// TwinCAT 3 PLC project Tc3_IoLink_Samples
// ProgramVersion: 3.1.4023.0
// libraries:
//   Tc2_Standard, * (Beckhoff Automation GmbH)
//   Tc2_System, * (Beckhoff Automation GmbH)
//   Tc3_IoLink, * (Beckhoff Automation GmbH)
//   Tc3_Module, * (Beckhoff Automation GmbH)
// project tree:
//   GVLs/ GVL_IO.TcGVL
//   / PlcTask.TcTTO
//   POUs/Samples/ FB_Sample_01_IolRead.TcPOU, FB_Sample_03_IolSlave.TcPOU, FB_Sample_02_IolWrite.TcPOU, FB_Sample_04_IolStdVarSlave.TcPOU, FB_Sample_06_IdentificationAndDiagnosis.TcPOU, FB_Sample_07_MeasurementDataChannel.TcPOU
//   POUs/ MAIN.TcPOU
// real-time tasks:
//   TASK PlcTask: cycle T#10ms, priority 20, ADS port 350
// I/O:
//   DEVICE Device 1 (EtherCAT), AmsNetId 192.168.178.79.2.1
//     Term 1 (EK1100) [EK1100 EtherCAT Coupler (2A E-Bus)]
//       Term 2 (EL6224) [EL6224 (IO Link Master)]
// variable links:
//   Tc3_IoLink_Samples/Tc3_IoLink_Samples Instance <-> Device 1 (EtherCAT)/Term 1 (EK1100)/Term 2 (EL6224)
//     PlcTask Inputs/GVL_IO.nTerm2Port{1..4}State <-> DeviceState Inputs/State Ch{1..4}  (4 links)
//     PlcTask Inputs/GVL_IO.sTerm2AmsNetId <-> InfoData/AoeNetId

CONFIGURATION Tc3_IoLink_Samples
    RESOURCE PLC ON TwinCAT3
        TASK PlcTask(INTERVAL := T#10ms, PRIORITY := 20);
        PROGRAM MAIN WITH PlcTask : MAIN;
    END_RESOURCE
END_CONFIGURATION

// ---- GVLs/GVL_IO.TcGVL
{attribute 'qualified_only'}
VAR_GLOBAL
	sTerm2AmsNetId 	AT%I*			: AMSNETID;
	
	nTerm2EPI1008					: E_IolPort := E_IolPort.Port1;
	nTerm2EPI2008					: E_IolPort := E_IolPort.Port2;
	nTerm2EPI3174					: E_IolPort := E_IolPort.Port3;

	nTerm2Port1State 	AT%I*		: USINT;
	nTerm2Port2State 	AT%I*		: USINT;
	nTerm2Port3State 	AT%I*		: USINT;
	nTerm2Port4State 	AT%I*		: USINT;
END_VAR

// ---- POUs/MAIN.TcPOU
PROGRAM MAIN
VAR
	fbSample_01_IolRead 					: FB_Sample_01_IolRead;
	fbSample_02_IolWrite 					: FB_Sample_02_IolWrite;
	fbSample_03_IolSlave 					: FB_Sample_03_IolSlave;
	fbSample_04_IolStdVarSlave 				: FB_Sample_04_IolStdVarSlave;
	fbSample_06_IdentificationAndDiagnosis	: FB_Sample_06_IdentificationAndDiagnosis;
	fbSample_07_MeasurementDataChannel		: FB_Sample_07_MeasurementDataChannel;
END_VAR


fbSample_01_IolRead(); 		
fbSample_02_IolWrite();	
fbSample_03_IolSlave(); 
fbSample_04_IolStdVarSlave();
fbSample_06_IdentificationAndDiagnosis();

END_PROGRAM

// ---- POUs/Samples/FB_Sample_01_IolRead.TcPOU
FUNCTION_BLOCK FB_Sample_01_IolRead
VAR_INPUT
	bExecute				: BOOL := FALSE;
END_VAR
VAR_OUTPUT
	bBusy					: BOOL := FALSE;
	bDone					: BOOL := FALSE;
	bError					: BOOL := FALSE;
	nAdsError				: E_AdsErr := E_AdsErr.NOERR;
	nIolError				: E_IolError := E_IolError.NoError;
	sErrorTxt				: STRING(255) := '';
	sApplicationTag			: STRING(32) := '';
END_VAR
VAR
	bExecuteOld				: BOOL;
	nState					: INT := 0;
	fbIolRead 				: FB_IolRead;
END_VAR

////
// Execute/Busy State Machine
//
IF bExecute AND NOT bExecuteOld AND NOT bBusy THEN
	bBusy := TRUE;
	nState := 10;	// READ
ELSIF NOT bExecute THEN
	bBusy := FALSE;
	bError := FALSE;
	bDone := FALSE;
	nAdsError := E_AdsErr.NOERR;
	nIolError := E_IolError.NoError;
	sErrorTxt := '';
END_IF
bExecuteOld := bExecute;

////
// FB State Machine
//
CASE nState OF
// IDLE
0:;
// READ
10:
	sApplicationTag := '';
	
	fbIolRead(bExecute := FALSE);
	fbIolRead.sNetId := F_CreateAmsNetId(GVL_IO.sTerm2AmsNetId);
	fbIolRead.nIolPort := E_IolPort.Port1;
	fbIolRead.pDSTBuf := ADR(sApplicationTag);
	fbIolRead.cbBufLen := 32;
	fbIolRead.nIndex := 16#18; 
	fbIolRead.nSubindex := 0;
	fbIolRead.bExecute := TRUE;
	
	nState := 20; // WAIT_FOR_DONE 
	
// WAIT_FOR_DONE
20:
	IF fbIolRead.bDone THEN
		bDone := TRUE;
		bBusy := FALSE;
		nState := 0; // IDLE
	END_IF 
END_CASE

////
// call FBs
//
fbIolRead();

////
// Error Handling
//
IF NOT bError AND bBusy THEN
	IF fbIolRead.bError THEN
		nState := 0;
		bBusy := FALSE;
		bError := TRUE;
		nAdsError := fbIolRead.nAdsError;
		nIolError := fbIolRead.nIolError;
		sErrorTxt := F_IolGetErrorTxt(fbIolRead.hresult);
	END_IF
END_IF

END_FUNCTION_BLOCK

// ---- POUs/Samples/FB_Sample_02_IolWrite.TcPOU
FUNCTION_BLOCK FB_Sample_02_IolWrite
VAR_INPUT
	bExecute				: BOOL := FALSE;
	sApplicationTag			: STRING(32) := '';
END_VAR
VAR_OUTPUT
	bBusy					: BOOL := FALSE;
	bDone					: BOOL := FALSE;
	bError					: BOOL := FALSE;
	nAdsError				: E_AdsErr := E_AdsErr.NOERR;
	nIolError				: E_IolError := E_IolError.NoError;
	sErrorTxt				: STRING(255) := '';
END_VAR
VAR
	bExecuteOld				: BOOL;
	nState					: INT := 0;
	fbIolWrite 				: FB_IolWrite;
END_VAR

////
// Execute/Busy State Machine
//
IF bExecute AND NOT bExecuteOld AND NOT bBusy THEN
	bBusy := TRUE;
	nState := 10;	// WRITE
ELSIF NOT bExecute THEN
	bBusy := FALSE;
	bError := FALSE;
	bDone := FALSE;
	nAdsError := E_AdsErr.NOERR;
	nIolError := E_IolError.NoError;
	sErrorTxt := '';
END_IF
bExecuteOld := bExecute;


////
// FB State Machine
//
CASE nState OF
	
// IDLE
0:;

// WRITE
10:	
	fbIolWrite(bExecute := FALSE);
	fbIolWrite.sNetId := F_CreateAmsNetId(GVL_IO.sTerm2AmsNetId);
	fbIolWrite.nIolPort := GVL_IO.nTerm2EPI1008;
	fbIolWrite.pSRCBuf := ADR(sApplicationTag);
	fbIolWrite.cbBufLen := 32;
	fbIolWrite.nIndex := 16#18;
	fbIolWrite.nSubindex := 0;
	fbIolWrite.bExecute := TRUE;
	
	nState := 20; // WAIT_FOR_DONE 
	
// WAIT_FOR_DONE
20:
	IF fbIolWrite.bDone THEN
		bDone := TRUE;
		bBusy := FALSE;
		nState := 0; // IDLE
	END_IF 
END_CASE


////
// call FBs
//
fbIolWrite();

////
// Error Handling
//
IF NOT bError AND bBusy THEN
	IF fbIolWrite.bError THEN
		nState := 0;
		bBusy := FALSE;
		bError := TRUE;
		nAdsError := fbIolWrite.nAdsError;
		nIolError := fbIolWrite.nIolError;
		sErrorTxt := F_IolGetErrorTxt(fbIolWrite.hresult);
	END_IF
END_IF

END_FUNCTION_BLOCK

// ---- POUs/Samples/FB_Sample_03_IolSlave.TcPOU
FUNCTION_BLOCK FB_Sample_03_IolSlave
VAR_INPUT
	bExecute				: BOOL := FALSE;
	sApplicationTag			: STRING(32) := '';
END_VAR
VAR_OUTPUT
	bBusy					: BOOL := FALSE;
	bDone					: BOOL := FALSE;
	bError					: BOOL := FALSE;
	nAdsError				: E_AdsErr := E_AdsErr.NOERR;
	nIolError				: E_IolError := E_IolError.NoError;
	sErrorTxt				: STRING(255) := '';
END_VAR
VAR
	bExecuteOld				: BOOL;
	nState					: INT := 0;
	fbIolSlave 				: FB_IolSlave;
	bInitDone				: BOOL := FALSE;
	hr						: HRESULT;
	sApplicationTagRead		: STRING(32) := '';
	sData					: STRING;
END_VAR

////
// Init
//
IF NOT bInitDone THEN
	bInitDone := TRUE;
	fbIolSlave.MasterAoeNetId := F_CreateAmsNetId(GVL_IO.sTerm2AmsNetId);
	fbIolSlave.Port := GVL_IO.nTerm2EPI1008;
	fbIolSlave.Name := 'EPI1008';
END_IF

////
// Execute/Busy State Machine
//
IF bExecute AND NOT bExecuteOld AND NOT bBusy THEN
	bBusy := TRUE;
	nState := 10;	// WRITE
ELSIF NOT bExecute THEN
	bBusy := FALSE;
	bError := FALSE;
	bDone := FALSE;
	nAdsError := E_AdsErr.NOERR;
	nIolError := E_IolError.NoError;
	sErrorTxt := '';
END_IF
bExecuteOld := bExecute;


////
// FB State Machine
//
CASE nState OF
	
// IDLE
0:;

// WRITE
10:
	hr := fbIolSlave.Write(16#0018, 0, ADR(sApplicationTag), 32);
	IF NOT F_IolIsBusy(hr) THEN
		IF FAILED(hr) THEN
			bBusy := FALSE;
			bError := TRUE;
			sErrorTxt := fbIolSlave.ErrorTxt;
			nAdsError := F_IolGetAdsError(hr);
			nIolError := F_IolGetIolError(hr);
			nState := 0; // IDLE;
		ELSE
			nState := 20; // READ;
		END_IF
	END_IF
	
// READ
20:
	hr := fbIolSlave.Read(16#0018, 16#00, ADR(sApplicationTagRead), 32);
	IF NOT F_IolIsBusy(hr) THEN
		IF FAILED(hr) THEN
			bBusy := FALSE;
			bError := TRUE;
			sErrorTxt := fbIolSlave.ErrorTxt;
			nAdsError := F_IolGetAdsError(hr);
			nIolError := F_IolGetIolError(hr);
			nState := 0; // IDLE;
		ELSE
			nState := 30; // CHECK;
		END_IF
	END_IF
	
// CHECK
30:
	IF sApplicationTag <> sApplicationTagRead THEN
		bBusy := FALSE;
		bError := TRUE;
		sErrorTxt := 'sApplicationTag and sApplicationTagRead are not equal!';
	ELSE
		bBusy := FALSE;
		bDone := TRUE;
		nState := 0;
	END_IF
END_CASE


////
// call FBs
//
fbIolSlave();

END_FUNCTION_BLOCK

// ---- POUs/Samples/FB_Sample_04_IolStdVarSlave.TcPOU
FUNCTION_BLOCK FB_Sample_04_IolStdVarSlave
VAR_INPUT
	bExecute				: BOOL := FALSE;
	sApplicationTag			: STRING(32) := '';
END_VAR
VAR_OUTPUT
	bBusy					: BOOL := FALSE;
	bDone					: BOOL := FALSE;
	bError					: BOOL := FALSE;
	nAdsError				: E_AdsErr := E_AdsErr.NOERR;
	nIolError				: E_IolError := E_IolError.NoError;
	sErrorTxt				: STRING(255) := '';
END_VAR
VAR
	bExecuteOld				: BOOL;
	nState					: INT := 0;
	fbIolSlave 				: FB_IolStdVarSlave;
	bInitDone				: BOOL := FALSE;
	hr						: HRESULT;
	sApplicationTagRead		: STRING(32) := '';
END_VAR

////
// Init
//
IF NOT bInitDone THEN
	bInitDone := TRUE;
	fbIolSlave.MasterAoeNetId := F_CreateAmsNetId(GVL_IO.sTerm2AmsNetId);
	fbIolSlave.Port := GVL_IO.nTerm2EPI1008;
	fbIolSlave.Name := 'EPI1008';
END_IF

////
// Execute/Busy State Machine
//
IF bExecute AND NOT bExecuteOld AND NOT bBusy THEN
	bBusy := TRUE;
	nState := 10;	// WRITE
ELSIF NOT bExecute THEN
	bBusy := FALSE;
	bError := FALSE;
	bDone := FALSE;
	nAdsError := E_AdsErr.NOERR;
	nIolError := E_IolError.NoError;
	sErrorTxt := '';
END_IF
bExecuteOld := bExecute;


////
// FB State Machine
//
CASE nState OF
	
// IDLE
0:;

// WRITE
10:
	hr := fbIolSlave.WriteApplicationSpecificTag(sApplicationTag);
	
	IF NOT F_IolIsBusy(hr) THEN
		IF FAILED(hr) THEN
			bBusy := FALSE;
			bError := TRUE;
			sErrorTxt := fbIolSlave.ErrorTxt;
			nAdsError := F_IolGetAdsError(hr);
			nIolError := F_IolGetIolError(hr);
			nState := 0; // IDLE;
		ELSE
			nState := 20; // READ;
		END_IF
	END_IF
	
// READ
20:
	hr := fbIolSlave.ReadApplicationSpecificTag(sApplicationTagRead);
	
	IF NOT F_IolIsBusy(hr) THEN
		IF FAILED(hr) THEN
			bBusy := FALSE;
			bError := TRUE;
			sErrorTxt := fbIolSlave.ErrorTxt;
			nAdsError := F_IolGetAdsError(hr);
			nIolError := F_IolGetIolError(hr);
			nState := 0; // IDLE;
		ELSE
			nState := 30; // CHECK;
		END_IF
	END_IF
	
// CHECK
30:
	IF sApplicationTag <> sApplicationTagRead THEN
		bBusy := FALSE;
		bError := TRUE;
		sErrorTxt := 'sApplicationTag and sApplicationTagRead are not equal!';
	ELSE
		bBusy := FALSE;
		bDone := TRUE;
		nState := 0;
	END_IF
END_CASE


////
// call FBs
//
fbIolSlave();

END_FUNCTION_BLOCK

// ---- POUs/Samples/FB_Sample_06_IdentificationAndDiagnosis.TcPOU
FUNCTION_BLOCK FB_Sample_06_IdentificationAndDiagnosis
VAR_INPUT
	sApplicationTagIn		: STRING(32) := '';
	sFunctionTagIn			: STRING(32) := '';
	sLocationTagIn			: STRING(32) := '';
	bExecute				: BOOL;
END_VAR
VAR_OUTPUT
	bBusy					: BOOL := FALSE;
	bDone					: BOOL := FALSE;
	bError					: BOOL := FALSE;
	
	sIolError				: STRING;
	sAdsError				: STRING;
	aProfileIDList			: ARRAY [0..31] OF E_IolProfileIdentifier;
	aFunctionClassIDList	: ARRAY[0..31] OF E_IolProfileIdentifier;
	stIDentObjects			: ST_IolIdentificationObjects;
	bDeviceOK				: BOOL;
	nDeviceStatus			: E_IolDeviceStatus;
	DetailedDeviceStatus	: T_IolDetailedDeviceStatus;
END_VAR
VAR
	bExecuteOld				: BOOL;
	nState					: INT := 0;
	IolDiagAndIdent			: IOL_IdentificationAndDiagnosis;
END_VAR

////
// Execute/Busy State Machine
//
IF bExecute AND NOT bExecuteOld AND NOT bBusy THEN
	bBusy := TRUE;
	nState := 10;	// START
ELSIF NOT bExecute THEN
	bBusy := FALSE;
	bError := FALSE;
	bDone := FALSE;
	sIolError:='';
	sADSError:='';
END_IF
bExecuteOld := bExecute;
	

CASE nState OF
	
// IDLE
0:;

// START
10:
	IolDiagAndIdent(Execute := FALSE);
	
	IolDiagAndIdent.MasterAoeNetId := F_CreateAmsNetId(GVL_IO.sTerm2AmsNetId);
	IolDiagAndIdent.IolPort := E_iolport.Port4;
	IolDiagAndIdent.Funct := E_IolIad_Function.ReadAll;
	IolDiagAndIdent.ApplicationSpecificTagIn := sApplicationTagIn;
	IolDiagAndIdent.FunctionTagIn := sFunctionTagIn;
	IolDiagAndIdent.LocationTagIn := sLocationTagIn;
	
	IolDiagAndIdent.Execute := TRUE;
	nState := 20; // WAIT FOR DONE
	
// WAIT FOR DONE
20:
	IF NOT IOlDiagAndIdent.Busy  AND NOT IOlDiagAndIdent.Error THEN 
		nState := 30; // DONE
	END_IF

// DONE
30:
	aProfileIDList := IolDiagAndIdent.ProfileIDList;
	aFunctionClassIDList := IolDiagAndIdent.FunctionClassIDList;
	stIDentObjects := IolDiagAndIdent.IdentificationObjects;
	bDeviceOK := IolDiagAndIdent.DeviceOK;
	nDeviceStatus := IolDiagAndIdent.DeviceStatus;
	DetailedDeviceStatus := IolDiagAndIdent.DetailedDeviceStatus;
	
	IolDiagAndIdent.Execute := FALSE;
	nState := 0; // INIT

END_CASE


////
// call FBs
//
IolDiagAndIdent();


////
// Error Handling
//
IF NOT bError AND bBusy THEN
	IF IolDiagAndIdent.Error THEN
		nState := 0;
		bBusy := FALSE;
		bError := TRUE;
		sIolError := F_IolGetIolErrorTxt(ioldiagandIdent.IolError);
		sAdsError := F_IolGetadsErrorTxt(ioldiagandident.AdsError);
	END_IF
END_IF

END_FUNCTION_BLOCK

// ---- POUs/Samples/FB_Sample_07_MeasurementDataChannel.TcPOU
FUNCTION_BLOCK FB_Sample_07_MeasurementDataChannel
VAR_INPUT
	nStateChannel		AT%I*	: USINT;
	nScale				AT%I*	: SINT;
	MVDistance			AT%I*	: INT;
END_VAR
VAR_OUTPUT
	bValid						: BOOL;
	bError						: BOOL;
	nValueStatus				: E_IolMdc_ValueStatus;
	nValueDINT					: DINT;
	nValueREAL					: LREAL;
	nScaleOut					: INT;
END_VAR
VAR
	fbMeasurement				: IOL_MeasurementDataChannel_INT;
END_VAR

fbMeasurement
(
	Enable := TRUE, 
	SubstituteValue := 500, 
	ChannelState := nStateChannel, 
	ScaleIn := nScale, 
	MeasurementValue := MVDistance, 
	Valid => bValid, 
	Error => bError, 
	ValueStatus => nValueStatus, 
	ValueReal => nValueREAL, 
	ValueDINT => nValueDINT, 
	Scale => nScaleOut 
);

END_FUNCTION_BLOCK
